// TwinCAT 3 PLC project MemRingBuffer
// ProgramVersion: 3.1.4024.0
// libraries:
//   Tc2_Standard, * (Beckhoff Automation GmbH)
//   Tc2_System, * (Beckhoff Automation GmbH)
//   Tc2_Utilities, * (Beckhoff Automation GmbH)
//   Tc3_Module, * (Beckhoff Automation GmbH)
// project tree:
//   DUTs/ E_EventType.TcDUT, ST_Event.TcDUT
//   / PlcTask.TcTTO
//   POUs/ FB_EventBuffer.TcPOU, MAIN.TcPOU

CONFIGURATION MemRingBuffer
    RESOURCE PLC ON TwinCAT3
        TASK PlcTask(INTERVAL := T#10ms, PRIORITY := 22);
        PROGRAM MAIN WITH PlcTask : MAIN;
    END_RESOURCE
END_CONFIGURATION

// ---- DUTs/E_EventType.TcDUT
{attribute 'qualified_only'}
{attribute 'strict'}
{attribute 'to_string'}
TYPE E_EventType :
(
	Alarm := 0,
	Message := 1
);
END_TYPE

// ---- DUTs/ST_Event.TcDUT
TYPE ST_Event :
STRUCT
	eEventType : E_EventType;
	eEventSeverity : TcEventSeverity;
	nEventIdentity : UDINT;
	sEventText : STRING(255);
	dtTimeStamp : DATE_AND_TIME;
END_STRUCT
END_TYPE

// ---- POUs/MAIN.TcPOU
PROGRAM MAIN
VAR
	EventBuffer : FB_EventBuffer;
	
	AddEvent : BOOL;
	stEventAdd : ST_Event;
	bErrorToAddEvent : BOOL;
	
	ReadAndRemoveEvent : BOOL;
	LastReadEvent : ST_Event;
	bErrorToReadRemoveEvent : BOOL;
	
END_VAR

IF AddEvent THEN
	EventBuffer.AddEvent(stEvent := stEventAdd, bError => bErrorToAddEvent);
	AddEvent := FALSE;
END_IF
IF ReadAndRemoveEvent THEN
	EventBuffer.GetRemoveEvent(stEvent => LastReadEvent, bError => bErrorToReadRemoveEvent);
	ReadAndRemoveEvent := FALSE;
END_IF

END_PROGRAM

// ---- POUs/FB_EventBuffer.TcPOU
FUNCTION_BLOCK FB_EventBuffer
VAR
	fbMemRingBuffer : FB_MemRingBuffer;
	BufferArray  : ARRAY[0..NUMBER_BYTES_FOR_ST_EVENT] OF BYTE; (* Buffer memory used by FB_MemRingBuffer function block *)
END_VAR

VAR CONSTANT
	ST_EVENT_SiZE : UDINT := SIZEOF(ST_Event); // size of a type
	MAX_NUMBER_ST_EVENT : UDINT := 5;
	NUMBER_BYTES_FOR_ST_EVENT : UDINT := MAX_NUMBER_ST_EVENT * ST_EVENT_SiZE;
END_VAR

METHOD PUBLIC AddEvent
VAR_INPUT
	stEvent : REFERENCE TO ST_Event;
END_VAR
VAR_OUTPUT
	bError : BOOL;
END_VAR
fbMemRingBuffer.A_AddTail(pWrite := ADR(stEvent),
							cbWrite := SIZEOF(stEvent),
							pBuffer := ADR(BufferArray),
							cbBuffer := SIZEOF(BufferArray));

bError := NOT fbMemRingBuffer.bOk;
END_METHOD

METHOD GetRemoveEvent
VAR_OUTPUT
	stEvent : ST_Event;
	bError : BOOL;
END_VAR
fbMemRingBuffer.A_RemoveHead(pRead := ADR(stEvent),
							cbRead := SIZEOF(stEvent),
							pBuffer := ADR(BufferArray),
							cbBuffer := SIZEOF(BufferArray));
							
bError := NOT fbMemRingBuffer.bOk;
END_METHOD

END_FUNCTION_BLOCK
